PROGRAM StnOverflowValveCtrl
VAR
END_VAR


IF bAutoPreparationPb AND ARbDI[Digital_Input.eX11013_Stn01ProcessTankSensor_Min_Overflow] AND ARbDO[eY10107_STN01PROCESSTANKPUMPON_OFF] THEN
ARwDO[eY13001_STN01OVERFLOWSUCTIONAV1_2].00 := TRUE;
ELSE
ARwDO[eY13001_STN01OVERFLOWSUCTIONAV1_2].00 := FALSE;	
END_IF


IF bAutoPreparationPb AND ARbDI[Digital_Input.eX11102_Stn03ProcessTankSensor_Min_Overflow] AND ARbDO[eY10109_STN03PROCESSTANKPUMPON_OFF] THEN
ARwDO[eY13004_STN03OVERFLOWSUCTIONAV3_2].00 := TRUE;
ELSE
ARwDO[eY13004_STN03OVERFLOWSUCTIONAV3_2].00 := FALSE;	
END_IF


IF bAutoPreparationPb AND ARbDI[Digital_Input.eX12006_Stn05ProcessTankSensor_Min_Overflow] AND ARbDO[eY10111_STN05PROCESSTANKPUMPON_OFF] THEN
ARwDO[eY13008_STN05OVERFLOWSUCTIONAV5_2].00 := TRUE;
ELSE
ARwDO[eY13008_STN05OVERFLOWSUCTIONAV5_2].00 := FALSE;	
END_IF

END_PROGRAM

(* stored: Version 1.1.0.1, ProductVersion 3.1.4024.12
   POU StnOverflowValveCtrl: Id {b2739bad-310c-4261-aac2-e338279dc2d1}, SpecialFunc None *)
